(* CODESYS project pile.export

Project tree, tasks and I/O mapping:
  pile/
    examples/
      program stack_examples [ST]
    function_blocks/
      function block stack [ST]: PEEK, POP, PUSH, is_empty, is_full
    object_models/
    visualisation/
      visualisation Visualization
*)

// pile/examples/stack_examples
PROGRAM stack_examples
VAR
	success	: BOOL;
	value : INT;
END_VAR

// Ajout d'une valeurs sur la pile
IF empiler_btn THEN
	success := my_stack.PUSH(element_value);
	empiler_btn := FALSE;
END_IF

// Retirer une valeur
IF depiler_btn THEN
	value := my_stack.POP();
	depiler_btn := FALSE;
END_IF;

END_PROGRAM

// pile/function_blocks/stack
FUNCTION_BLOCK stack

VAR CONSTANT
	MAX_SIZE :		INT							:= 10;		// Taille maximale de la pile
END_VAR

VAR
	stackArray : 	ARRAY[1..MAX_SIZE] OF INT	;			// Tableau pour stocker les éléments
	top :			INT							:= 0; 		// Indice du sommet de la pile
	errorCode :		INT							:= 0;		// Code d'erreur : 0 -> OK, 1 -> Overflow (Débordement), 2 -> Underflow (Vide)
END_VAR

// PUSH		: Méthode pour ajouter un élément au sommet de la pile.
// POP  	: Méthode pour retirer l'élément au sommet de la pile.
// PEEK		: Méthode pour connaitre la valeur de l'élément au sommet de la pile.

// is_empty : Propriété qui définie si la pile est vide.
// is_full	: Propriété qui définie si la pile est pleine.

METHOD PEEK : INT
VAR_INPUT
END_VAR
PEEK := 0;
errorCode := 0; 	// Réinitialisation du code d'erreur.

IF top > 0 THEN
    PEEK := stackArray[top];
ELSE
    errorCode := 2; // Erreur : Pile vide (Underflow)
END_IF;
END_METHOD

METHOD POP : INT
VAR_INPUT
END_VAR
POP := 0;
errorCode := 0; 	// Réinitialisation du code d'erreur.

IF top > 0 THEN
	POP := stackArray[top];
	top := top - 1;
ELSE
	errorCode := 2;	// Erreur : Pile vide (Underflow).
END_IF
END_METHOD

METHOD PUSH : BOOL
VAR_INPUT
	value	: INT;
END_VAR
PUSH := FALSE;
errorCode := 0;		// Réinitialisation du code d'erreur.

IF top < MAX_SIZE THEN
	top := top + 1;
	stackArray[top] := value;
	PUSH := TRUE;
ELSE
	errorCode := 1;	// Erreur : Dépassement de la pile (Overflow).
END_IF
END_METHOD

PROPERTY is_empty : BOOL
GET
is_empty := top = 0;
END_GET
SET
END_SET
END_PROPERTY

PROPERTY is_full : BOOL
GET
is_full := top = MAX_SIZE;
END_GET
SET
END_SET
END_PROPERTY

END_FUNCTION_BLOCK

// pile/visualisation/Visualization
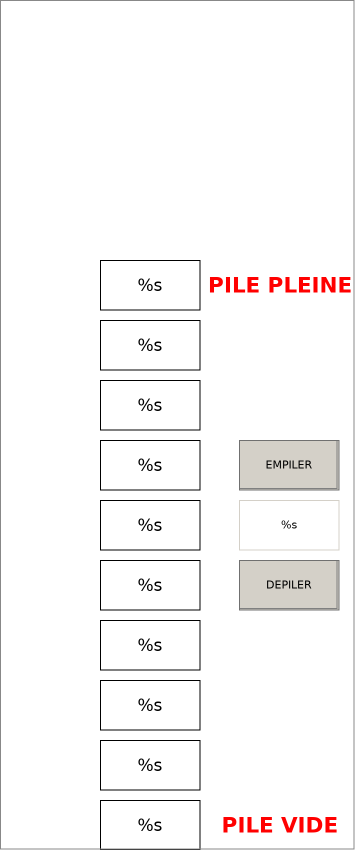
VISUALIZATION Visualization  // 355x850
    Rectangle (100,800 100x50), "%s", text variable: my_stack.stackArray[1], invisible if: my_stack.top<1
    Rectangle (100,740 100x50), "%s", text variable: my_stack.stackArray[2], invisible if: my_stack.top<2
    Rectangle (100,680 100x50), "%s", text variable: my_stack.stackArray[3], invisible if: my_stack.top<3
    Rectangle (100,620 100x50), "%s", text variable: my_stack.stackArray[4], invisible if: my_stack.top<4
    Rectangle (100,560 100x50), "%s", text variable: my_stack.stackArray[5], invisible if: my_stack.top<5
    Rectangle (100,500 100x50), "%s", text variable: my_stack.stackArray[6], invisible if: my_stack.top<6
    Rectangle (100,440 100x50), "%s", text variable: my_stack.stackArray[7], invisible if: my_stack.top<7
    Rectangle (100,380 100x50), "%s", text variable: my_stack.stackArray[8], invisible if: my_stack.top<8
    Rectangle (100,320 100x50), "%s", text variable: my_stack.stackArray[9], invisible if: my_stack.top<9
    Rectangle (100,260 100x50), "%s", text variable: my_stack.stackArray[10], invisible if: my_stack.top<10
    Label (205,810 150x30), "PILE VIDE", invisible if: NOT my_stack.is_empty
    Label (205,270 150x30), "PILE PLEINE", invisible if: NOT my_stack.is_full
    Button (239,440 100x50), "EMPILER"
        OnMouseClick:  ToggleVariable=empiler_btn
    Button (239,560 100x50), "DEPILER"
        OnMouseClick:  ToggleVariable=depiler_btn
    Textfield (239,500 100x50), "%s", text variable: element_value
        OnMouseClick: write the text variable via Default
END_VISUALIZATION
